(* This function block is created for interface devices between different PLC*)
(* Not all the Variables in the original structure is required, just few signals *)
(* They have to be linked to the custom created variables on the EL6692/5 primary side*)
FUNCTION_BLOCK FB_PIP_Interface_Out
VAR_INPUT
	VG : ST_VG;
END_VAR
VAR_OUTPUT
END_VAR
VAR
	i_rPRESS AT%Q*: REAL; 
	i_xAT_VAC AT%Q*: BOOL;
	i_xPRESS_OK AT%Q*: BOOL;
END_VAR

(* This function block is created for interface devices between different PLC*)
(* Not all the Variables in the original structure is required, just few signals *)
(* They have to be linked to the custom created variables on the EL6692/5 primary side*)

i_rPRESS:=VG.rPRESS;
i_xAT_VAC:= VG.xAT_VAC;
i_xPRESS_OK:=VG.xPRESS_OK;

END_FUNCTION_BLOCK

(* stored: Version 1.1.0.1, ProductVersion 3.1.4022.18
   POU FB_PIP_Interface_Out: Id {4731aeb7-0beb-4e3d-84b8-834f411d3c2f}, SpecialFunc None *)
